// TIA Portal V15.1 export
// export: Created 2024-05-17T05:38:20.2677605Z, ExportSetting WithDefaults, DisplayName Totally Integrated Automation Portal, DisplayVersion V15.1 Update 5, DisplayName TIA Portal Openness, DisplayVersion V15.1 Update 5, DisplayName SINAMICS Startdrive Advanced, DisplayVersion V15.1, DisplayName G130, G150, S120, S150, SINAMICS MV, S210, DisplayVersion V15.1, DisplayName G110M, G120, G120C, G120D, G120P, DisplayVersion V15.1, DisplayName STEP 7 Professional, DisplayVersion V15.1 Update 5, DisplayName STEP 7 Safety, DisplayVersion V15.1, DisplayName WinCC Professional, DisplayVersion V15.1 Update 5, DisplayName SIMATIC Visualization Architect, DisplayVersion V15.1
DATA_BLOCK "_209220ZM01Andon"   // DB356
{ S7_Optimized_Access := 'FALSE' }
AUTHOR : VCG
VERSION : 0.1
// stored: AutoNumber false, DBAccessibleFromOPCUA true, IsOnlyStoredInLoadMemory false, IsWriteProtectedInAS false
   VAR RETAIN
      AlarmA { ExternalAccessible := 'False'; ExternalVisible := 'False'; ExternalWritable := 'False'} : Bool;   // Summary Alarm A
      AlarmB { ExternalAccessible := 'False'; ExternalVisible := 'False'; ExternalWritable := 'False'} : Bool;   // Summary Alarm B
      AlarmC { ExternalAccessible := 'False'; ExternalVisible := 'False'; ExternalWritable := 'False'} : Bool;   // Summary Alarm C
      AlarmD { ExternalAccessible := 'False'; ExternalVisible := 'False'; ExternalWritable := 'False'} : Bool;   // Summary Alarm D
      AlarmABCondition { ExternalAccessible := 'False'; ExternalVisible := 'False'; ExternalWritable := 'False'} : Bool;   // Alarm AB condition
      H_Anim : Word;   // Animation
      H_DBnr : Int;   // DB number
      H_HMICmd : Word;   // HMI Command
      H_HMI : Struct   // Icon Animation
         AndonReq : "H_HMI";   // HMI Animation of the icon
         "209220CWP11SH01AndonHCall" : "H_HMI";   // HMI Animation of the icon
         "209220CWP12SH01AndonHCall" : "H_HMI";   // HMI Animation of the icon
         "209220CWP13SH01AndonHCall" : "H_HMI";   // HMI Animation of the icon
         "209220CWP14SH01AndonHCall" : "H_HMI";   // HMI Animation of the icon
         "209220CWP15SH01AndonHCall" : "H_HMI";   // HMI Animation of the icon
         "209220CWP16SH01AndonHCall" : "H_HMI";   // HMI Animation of the icon
         "209220CWP21SH01AndonHCall" : "H_HMI";   // HMI Animation of the icon
         "209220CWP22SH01AndonHCall" : "H_HMI";   // HMI Animation of the icon
         "209220CWP23SH01AndonHCall" : "H_HMI";   // HMI Animation of the icon
         "209220CWP24SH01AndonHCall" : "H_HMI";   // HMI Animation of the icon
         "209220CWP25SH01AndonHCall" : "H_HMI";   // HMI Animation of the icon
         "209220CWP26SH01AndonHCall" : "H_HMI";   // HMI Animation of the icon
      END_STRUCT;
      H : Struct   // Animation
         AndonReq : "H_AndonReqVCG";   // HMI Animation
         "209220CWP11SH01AndonHCall" : "H_GBAndonHCall";   // HMI Animation
         "209220CWP12SH01AndonHCall" : "H_GBAndonHCall";   // HMI Animation
         "209220CWP13SH01AndonHCall" : "H_GBAndonHCall";   // HMI Animation
         "209220CWP14SH01AndonHCall" : "H_GBAndonHCall";   // HMI Animation
         "209220CWP15SH01AndonHCall" : "H_GBAndonHCall";   // HMI Animation
         "209220CWP16SH01AndonHCall" : "H_GBAndonHCall";   // HMI Animation
         "209220CWP21SH01AndonHCall" : "H_GBAndonHCall";   // HMI Animation
         "209220CWP22SH01AndonHCall" : "H_GBAndonHCall";   // HMI Animation
         "209220CWP23SH01AndonHCall" : "H_GBAndonHCall";   // HMI Animation
         "209220CWP24SH01AndonHCall" : "H_GBAndonHCall";   // HMI Animation
         "209220CWP25SH01AndonHCall" : "H_GBAndonHCall";   // HMI Animation
         "209220CWP26SH01AndonHCall" : "H_GBAndonHCall";   // HMI Animation
      END_STRUCT;
      AndonStatus { ExternalAccessible := 'False'; ExternalVisible := 'False'; ExternalWritable := 'False'} : "AndonStatusVCG";   // Status
      AndonDataExchange { ExternalAccessible := 'False'; ExternalVisible := 'False'; ExternalWritable := 'False'} : "AndonDataExchangeVCG";   // Data Exchange
      AndonHCall { ExternalAccessible := 'False'; ExternalVisible := 'False'; ExternalWritable := 'False'} : Array[1..32] of Bool;   // Andon Human Call (Cycle Stop)
      AndonHCall_209220CWP11 { ExternalAccessible := 'False'; ExternalVisible := 'False'; ExternalWritable := 'False'} : Bool;   // Human Call
      AndonHCall_209220CWP12 { ExternalAccessible := 'False'; ExternalVisible := 'False'; ExternalWritable := 'False'} : Bool;   // Human Call
      AndonHCall_209220CWP13 { ExternalAccessible := 'False'; ExternalVisible := 'False'; ExternalWritable := 'False'} : Bool;   // Human Call
      AndonHCall_209220CWP14 { ExternalAccessible := 'False'; ExternalVisible := 'False'; ExternalWritable := 'False'} : Bool;   // Human Call
      AndonHCall_209220CWP15 { ExternalAccessible := 'False'; ExternalVisible := 'False'; ExternalWritable := 'False'} : Bool;   // Human Call
      AndonHCall_209220CWP16 { ExternalAccessible := 'False'; ExternalVisible := 'False'; ExternalWritable := 'False'} : Bool;   // Human Call
      AndonHCall_209220CWP21 { ExternalAccessible := 'False'; ExternalVisible := 'False'; ExternalWritable := 'False'} : Bool;   // Human Call
      AndonHCall_209220CWP22 { ExternalAccessible := 'False'; ExternalVisible := 'False'; ExternalWritable := 'False'} : Bool;   // Human Call
      AndonHCall_209220CWP23 { ExternalAccessible := 'False'; ExternalVisible := 'False'; ExternalWritable := 'False'} : Bool;   // Human Call
      AndonHCall_209220CWP24 { ExternalAccessible := 'False'; ExternalVisible := 'False'; ExternalWritable := 'False'} : Bool;   // Human Call
      AndonHCall_209220CWP25 { ExternalAccessible := 'False'; ExternalVisible := 'False'; ExternalWritable := 'False'} : Bool;   // Human Call
      AndonHCall_209220CWP26 { ExternalAccessible := 'False'; ExternalVisible := 'False'; ExternalWritable := 'False'} : Bool;   // Human Call
      AndonStopReqHCall { ExternalAccessible := 'False'; ExternalVisible := 'False'; ExternalWritable := 'False'} : Bool;   // Stop Request by Andon Human Call / Stop request - from dataPLC
   END_VAR
BEGIN
END_DATA_BLOCK
